TYPE ResponseData : 
STRUCT
	Header : STRING(Constants.HEADER_STRING_SIZE);
	Payload : STRING(Constants.PAYLOAD_STRING_SIZE);
END_STRUCT
END_TYPE

(* stored: Version 1.1.0.1, ProductVersion 3.1.4024.12
   DUT ResponseData: Id {9f3087a2-4dcc-4a26-a54b-d846ba814219} *)
